(* CODESYS project xlh_gantry_00_01.project
   Description: Receives some incoming messages and echoes them with CAN-ID +1
   Company: 3S - Smart Software Solutions GmbH
   Version: 1.0.0.0
   Title: CAN Bus API Example
   Author: 3S - Smart Software Solutions GmbH

Project tree, tasks and I/O mapping:
  xLH_base : CODESYS Control for Raspberry Pi 64 SL, CODESYS, order no. 2302000009, version 4.18.0.0
    application app
      libraries: Standard, 3.5.18.0 (System); Util, 3.5.21.0 (System); VisuDialogs, * (System); Memory, * (3S - Smart Software Solutions GmbH); CmpBitmapPool, * (System); CAN API, 1.0.0.4 (CODESYS); MemoryUtils, * (3S - Smart Software Solutions GmbH); CAA CiA 405, 4.3.0.0 (CODESYS)
      task CAN_OPEN_TASK (cyclic, interval 1 ms, priority 0) calls nothing
      task VISU_TASK (cyclic, interval 100 ms, priority 31) calls VisuElems.Visu_Prg
      task MAIN_TASK (cyclic, interval 4 ms, priority 1) calls io, MAIN_CALLER
      task SoftMotion_PlanningTask (cyclic, interval t#2ms, priority 15) calls nothing
      program MAIN_CALLER [ST]
      function block FB_SDO_READ_4_BYTE [ST]
      trace Trace_AxY (task MAIN_TASK): y_axis.fActPosition, y_axis.fSetPosition, y_axis.fSetAcceleration, y_axis.fActAcceleration, y_axis.fSetVelocity, y_axis.fActVelocity
      visualisation Visualization
      trace Trace (task MAIN_TASK): MC.diPosition, MC.iSetSpeed, MC.iDebug2Pos, MC.iDebug1Mileage, MC.auiUltrasonic[1], MC.fbReadStatusLoopTime.udiValue, MC.iSpeed2, MC.iSpeed1, MC.iPitch
      data type MOTION_CONTROL_BYTE
      MOTION_BASE/
        function block FB_XLH_MOTION_AXIS_SIMPLE_ES [ST]: mRead
        function block FB_PLC_OPEN_AXIS [ST]: plcOpen, executeToFalse
        function block FB_XLH_MOTION_AXIS_SIMPLE [ST]
        function block FB_XLH_MOTION_AXIS_BASE [ST]: mRead, mWrite
      IO/
        function block FB_XLH_GPIO [CFC]
        program io [ST]
        function block FB_XLH_DXL_RGB [CFC]
      program MC [ST]: write, read, axSmExecuteToFalse
      axis group AxisGroup: TRAFO.Kin_Gantry3, axes x_axis, y_axis, z_axis
    CANbus : CANbus, CODESYS, version 4.3.0.0
        settings: Baudrate = 1000 kbit/s
      CANopen_Manager : CANopen_Manager, CODESYS, version 4.3.0.0
          settings: NMT Start All = TRUE; Polling of optional slaves = FALSE; ConfigVersion = 50659584
        xlh_dynamixel_rgb : xlh_stamp_dynamixel_rgb, xemax ag, order no. 0, version Revision=16#00000001, FileVersion=1.0 (disabled)
            settings: NODEIDSAVED = 2; SDO Timeout = 1000000; PDO_Autoconfig = FALSE; EXPERTSETTINGS = FALSE; PDO 16#1400.COBID = 16#00000202; Process by CANopenManager = TRUE; PDO 16#1401.COBID = 16#00000302; Process by CANopenManager = TRUE; PDO 16#1402.COBID = 16#00000402; Process by CANopenManager = TRUE; PDO 16#1800.COBID = 16#00000182; Process by CANopenManager = TRUE; Dxl 1 Control.Subindex = 16#01; Dxl 1 Position.Subindex = 16#02; Dxl 1 Velocity.Subindex = 16#03; Dxl 2 Control.Subindex = 16#04; Dxl 2 Position.Subindex = 16#05; Dxl 2 Velocity.Subindex = 16#06; RGB red.Subindex = 16#01; RGB green.Subindex = 16#02; RGB blue.Subindex = 16#03; Dxl 1  Position read.Subindex = 16#01; Dxl 1 Current read.Subindex = 16#02; Dxl 2  Position read.Subindex = 16#03; Dxl 2 Current read.Subindex = 16#04; SDO List.Set COB-ID sync.Index = 16#1005; SDO List.Set COB-ID sync.Subindex = 16#00; SDO List.Set COB-ID sync.Value = 16#00000080; SDO List.Set COB-ID sync.Size = 32; SDO List.Set COB-ID sync.AbortIfError = FALSE; SDO List.Set COB-ID sync.JumpToLine = FALSE; SDO List.Set COB-ID sync.Line = 0; SDO List.Set communication cycle period.Index = 16#1006; SDO List.Set communication cycle period.Subindex = 16#00; SDO List.Set communication cycle period.Value = 16#00000000; SDO List.Set communication cycle period.Size = 32; SDO List.Set communication cycle period.AbortIfError = FALSE; SDO List.Set communication cycle period.JumpToLine = FALSE; SDO List.Set communication cycle period.Line = 0; SDO List.Set Guardtime.Index = 16#100C;
              SDO List.Set Guardtime.Subindex = 16#00; SDO List.Set Guardtime.Value = 16#000000C8; SDO List.Set Guardtime.Size = 16; SDO List.Set Guardtime.AbortIfError = FALSE; SDO List.Set Guardtime.JumpToLine = FALSE; SDO List.Set Guardtime.Line = 0; SDO List.Set Lifetime.Index = 16#100D; SDO List.Set Lifetime.Subindex = 16#00; SDO List.Set Lifetime.Value = 16#00000003; SDO List.Set Lifetime.Size = 8; SDO List.Set Lifetime.AbortIfError = FALSE; SDO List.Set Lifetime.JumpToLine = FALSE; SDO List.Set Lifetime.Line = 0; SDO List.Set Heartbeat Consumer.Index = 16#1016; SDO List.Set Heartbeat Consumer.Subindex = 16#01; SDO List.Set Heartbeat Consumer.Value = 0; SDO List.Set Heartbeat Consumer.Size = 32; SDO List.Set Heartbeat Consumer.AbortIfError = FALSE; SDO List.Set Heartbeat Consumer.JumpToLine = FALSE; SDO List.Set Heartbeat Consumer.Line = 0; SDO List.Disable PDO.Index = 16#1400; SDO List.Disable PDO.Subindex = 16#01; SDO List.Disable PDO.Value = 16#80000202; SDO List.Disable PDO.Size = 32; SDO List.Disable PDO.AbortIfError = FALSE; SDO List.Disable PDO.JumpToLine = FALSE; SDO List.Disable PDO.Line = 0; SDO List.Set transmission type.Index = 16#1400; SDO List.Set transmission type.Subindex = 16#02; SDO List.Set transmission type.Value = 16#FF; SDO List.Set transmission type.Size = 8; SDO List.Set transmission type.AbortIfError = FALSE; SDO List.Set transmission type.JumpToLine = FALSE; SDO List.Set transmission type.Line = 0; SDO List.Set and enable COB-ID.Index = 16#1400; SDO List.Set and enable COB-ID.Subindex = 16#01; SDO List.Set and enable COB-ID.Value = 16#00000202; SDO List.Set and enable COB-ID.Size = 32; SDO List.Set and enable COB-ID.AbortIfError = FALSE; SDO List.Set and enable COB-ID.JumpToLine = FALSE;
              SDO List.Set and enable COB-ID.Line = 0; SDO List.Disable PDO.Index = 16#1401; SDO List.Disable PDO.Subindex = 16#01; SDO List.Disable PDO.Value = 16#80000302; SDO List.Disable PDO.Size = 32; SDO List.Disable PDO.AbortIfError = FALSE; SDO List.Disable PDO.JumpToLine = FALSE; SDO List.Disable PDO.Line = 0; SDO List.Set transmission type.Index = 16#1401; SDO List.Set transmission type.Subindex = 16#02; SDO List.Set transmission type.Value = 16#FF; SDO List.Set transmission type.Size = 8; SDO List.Set transmission type.AbortIfError = FALSE; SDO List.Set transmission type.JumpToLine = FALSE; SDO List.Set transmission type.Line = 0; SDO List.Set and enable COB-ID.Index = 16#1401; SDO List.Set and enable COB-ID.Subindex = 16#01; SDO List.Set and enable COB-ID.Value = 16#00000302; SDO List.Set and enable COB-ID.Size = 32; SDO List.Set and enable COB-ID.AbortIfError = FALSE; SDO List.Set and enable COB-ID.JumpToLine = FALSE; SDO List.Set and enable COB-ID.Line = 0; SDO List.Disable PDO.Index = 16#1402; SDO List.Disable PDO.Subindex = 16#01; SDO List.Disable PDO.Value = 16#80000402; SDO List.Disable PDO.Size = 32; SDO List.Disable PDO.AbortIfError = FALSE; SDO List.Disable PDO.JumpToLine = FALSE; SDO List.Disable PDO.Line = 0; SDO List.Set transmission type.Index = 16#1402; SDO List.Set transmission type.Subindex = 16#02; SDO List.Set transmission type.Value = 16#FF; SDO List.Set transmission type.Size = 8; SDO List.Set transmission type.AbortIfError = FALSE; SDO List.Set transmission type.JumpToLine = FALSE; SDO List.Set transmission type.Line = 0; SDO List.Set and enable COB-ID.Index = 16#1402; SDO List.Set and enable COB-ID.Subindex = 16#01; SDO List.Set and enable COB-ID.Value = 16#00000402; SDO List.Set and enable COB-ID.Size = 32;
              SDO List.Set and enable COB-ID.AbortIfError = FALSE; SDO List.Set and enable COB-ID.JumpToLine = FALSE; SDO List.Set and enable COB-ID.Line = 0; SDO List.Disable PDO.Index = 16#1800; SDO List.Disable PDO.Subindex = 16#01; SDO List.Disable PDO.Value = 16#80000182; SDO List.Disable PDO.Size = 32; SDO List.Disable PDO.AbortIfError = FALSE; SDO List.Disable PDO.JumpToLine = FALSE; SDO List.Disable PDO.Line = 0; SDO List.Set transmission type.Index = 16#1800; SDO List.Set transmission type.Subindex = 16#02; SDO List.Set transmission type.Value = 16#FF; SDO List.Set transmission type.Size = 8; SDO List.Set transmission type.AbortIfError = FALSE; SDO List.Set transmission type.JumpToLine = FALSE; SDO List.Set transmission type.Line = 0; SDO List.Set inhibit time.Index = 16#1800; SDO List.Set inhibit time.Subindex = 16#03; SDO List.Set inhibit time.Value = 16#0000; SDO List.Set inhibit time.Size = 16; SDO List.Set inhibit time.AbortIfError = FALSE; SDO List.Set inhibit time.JumpToLine = FALSE; SDO List.Set inhibit time.Line = 0; SDO List.Set event time.Index = 16#1800; SDO List.Set event time.Subindex = 16#05; SDO List.Set event time.Value = 16#0000; SDO List.Set event time.Size = 16; SDO List.Set event time.AbortIfError = FALSE; SDO List.Set event time.JumpToLine = FALSE; SDO List.Set event time.Line = 0; SDO List.Set and enable COB-ID.Index = 16#1800; SDO List.Set and enable COB-ID.Subindex = 16#01; SDO List.Set and enable COB-ID.Value = 16#00000182; SDO List.Set and enable COB-ID.Size = 32; SDO List.Set and enable COB-ID.AbortIfError = FALSE; SDO List.Set and enable COB-ID.JumpToLine = FALSE; SDO List.Set and enable COB-ID.Line = 0; ConfigVersion = 50659584
            output app.io.dxlRgb.bDxl1Torque : BOOL  // Dxl 1 Control.Bit0
            output app.io.dxlRgb.bDxl1Led : BOOL  // Dxl 1 Control.Bit1
            output app.io.dxlRgb.uiDxl1Position : UINT  // Dxl 1 Position
            output app.io.dxlRgb.uiDxl1Velocity : UINT  // Dxl 1 Velocity
            output app.io.dxlRgb.bDxl2Torque : BOOL  // Dxl 2 Control.Bit0
            output app.io.dxlRgb.bDxl2Led : BOOL  // Dxl 2 Control.Bit1
            output app.io.dxlRgb.uiDxl2Position : UINT  // Dxl 2 Position
            output app.io.dxlRgb.uiDxl2Velocity : UINT  // Dxl 2 Velocity
            output app.io.dxlRgb.byRgbRed : USINT  // RGB red
            output app.io.dxlRgb.byRgbGreen : USINT  // RGB green
            output app.io.dxlRgb.byRgbBlue : USINT  // RGB blue
            input  app.io.dxlRgb.uiDxl1PositionGet : UINT  // Dxl 1  Position read
            input  app.io.dxlRgb.iDxl1CurrentGet : INT  // Dxl 1 Current read
            input  app.io.dxlRgb.uiDxl2PositionGet : UINT  // Dxl 2  Position read
            input  app.io.dxlRgb.iDxl2CurrentGet : INT  // Dxl 2 Current read
            unmapped channels: Dxl 1 Control, Dxl 2 Control
        xlh_motion : xlh_motion, xemax ag, order no. 0, version Revision=16#00000001, FileVersion=1.0
            settings: NODEIDSAVED = 1; SDO Timeout = 1000000; PDO_Autoconfig = FALSE; EXPERTSETTINGS = True; PDO 16#1400.COBID = 16#00000201; Process by CANopenManager = TRUE; PDO 16#1401.COBID = 16#00000301; Process by CANopenManager = TRUE; PDO 16#1402.COBID = 16#00000401; Process by CANopenManager = TRUE; PDO 16#1403.COBID = 16#00000501; Process by CANopenManager = TRUE; PDO 16#1800.COBID = 16#00000181; Process by CANopenManager = TRUE; PDO 16#1801.COBID = 16#00000281; Process by CANopenManager = TRUE; PDO 16#1802.COBID = 16#00000381; Process by CANopenManager = TRUE; Control 1.Subindex = 16#01; Control 2.Subindex = 16#02; Control 3.Subindex = 16#03; Control 4.Subindex = 16#04; Outputs 0-7.Subindex = 16#01; Outputs 8-15.Subindex = 16#02; Magnet Duty Cycle.Subindex = 16#01; Freqeuncy 1.Subindex = 16#05; Freqeuncy 2.Subindex = 16#06; Freqeuncy 3.Subindex = 16#07; Freqeuncy 4.Subindex = 16#08; Servo 1.Subindex = 16#01; Servo 2.Subindex = 16#02; Servo 3.Subindex = 16#03; Servo 4.Subindex = 16#04; Servo 5.Subindex = 16#05; Servo 6.Subindex = 16#06; Servo 7.Subindex = 16#07; Servo 8.Subindex = 16#08; Position 1.Subindex = 16#01; Position 2.Subindex = 16#02; Position 3.Subindex = 16#03;
              Position 4.Subindex = 16#04; Inputs 0-7.Subindex = 16#01; Inputs 8-15.Subindex = 16#02; Inputs CLK.Subindex = 16#03; SDO List.Set COB-ID sync.Index = 16#1005; SDO List.Set COB-ID sync.Subindex = 16#00; SDO List.Set COB-ID sync.Value = 16#00000080; SDO List.Set COB-ID sync.Size = 32; SDO List.Set COB-ID sync.AbortIfError = FALSE; SDO List.Set COB-ID sync.JumpToLine = FALSE; SDO List.Set COB-ID sync.Line = 0; SDO List.Set communication cycle period.Index = 16#1006; SDO List.Set communication cycle period.Subindex = 16#00; SDO List.Set communication cycle period.Value = 16#00000000; SDO List.Set communication cycle period.Size = 32; SDO List.Set communication cycle period.AbortIfError = FALSE; SDO List.Set communication cycle period.JumpToLine = FALSE; SDO List.Set communication cycle period.Line = 0; SDO List.Set Guardtime.Index = 16#100C; SDO List.Set Guardtime.Subindex = 16#00; SDO List.Set Guardtime.Value = 16#000000C8; SDO List.Set Guardtime.Size = 16; SDO List.Set Guardtime.AbortIfError = FALSE; SDO List.Set Guardtime.JumpToLine = FALSE; SDO List.Set Guardtime.Line = 0; SDO List.Set Lifetime.Index = 16#100D; SDO List.Set Lifetime.Subindex = 16#00; SDO List.Set Lifetime.Value = 16#00000003; SDO List.Set Lifetime.Size = 8; SDO List.Set Lifetime.AbortIfError = FALSE; SDO List.Set Lifetime.JumpToLine = FALSE; SDO List.Set Lifetime.Line = 0; SDO List.Set Heartbeat Consumer.Index = 16#1016; SDO List.Set Heartbeat Consumer.Subindex = 16#01; SDO List.Set Heartbeat Consumer.Value = 0; SDO List.Set Heartbeat Consumer.Size = 32; SDO List.Set Heartbeat Consumer.AbortIfError = FALSE; SDO List.Set Heartbeat Consumer.JumpToLine = FALSE; SDO List.Set Heartbeat Consumer.Line = 0; SDO List.Disable PDO.Index = 16#1400;
              SDO List.Disable PDO.Subindex = 16#01; SDO List.Disable PDO.Value = 16#80000201; SDO List.Disable PDO.Size = 32; SDO List.Disable PDO.AbortIfError = FALSE; SDO List.Disable PDO.JumpToLine = FALSE; SDO List.Disable PDO.Line = 0; SDO List.Set transmission type.Index = 16#1400; SDO List.Set transmission type.Subindex = 16#02; SDO List.Set transmission type.Value = 16#FF; SDO List.Set transmission type.Size = 8; SDO List.Set transmission type.AbortIfError = FALSE; SDO List.Set transmission type.JumpToLine = FALSE; SDO List.Set transmission type.Line = 0; SDO List.Set and enable COB-ID.Index = 16#1400; SDO List.Set and enable COB-ID.Subindex = 16#01; SDO List.Set and enable COB-ID.Value = 16#00000201; SDO List.Set and enable COB-ID.Size = 32; SDO List.Set and enable COB-ID.AbortIfError = FALSE; SDO List.Set and enable COB-ID.JumpToLine = FALSE; SDO List.Set and enable COB-ID.Line = 0; SDO List.Disable PDO.Index = 16#1401; SDO List.Disable PDO.Subindex = 16#01; SDO List.Disable PDO.Value = 16#80000301; SDO List.Disable PDO.Size = 32; SDO List.Disable PDO.AbortIfError = FALSE; SDO List.Disable PDO.JumpToLine = FALSE; SDO List.Disable PDO.Line = 0; SDO List.Set transmission type.Index = 16#1401; SDO List.Set transmission type.Subindex = 16#02; SDO List.Set transmission type.Value = 16#FF; SDO List.Set transmission type.Size = 8; SDO List.Set transmission type.AbortIfError = FALSE; SDO List.Set transmission type.JumpToLine = FALSE; SDO List.Set transmission type.Line = 0; SDO List.Set and enable COB-ID.Index = 16#1401; SDO List.Set and enable COB-ID.Subindex = 16#01; SDO List.Set and enable COB-ID.Value = 16#00000301; SDO List.Set and enable COB-ID.Size = 32; SDO List.Set and enable COB-ID.AbortIfError = FALSE; SDO List.Set and enable COB-ID.JumpToLine = FALSE;
              SDO List.Set and enable COB-ID.Line = 0; SDO List.Disable PDO.Index = 16#1402; SDO List.Disable PDO.Subindex = 16#01; SDO List.Disable PDO.Value = 16#80000401; SDO List.Disable PDO.Size = 32; SDO List.Disable PDO.AbortIfError = FALSE; SDO List.Disable PDO.JumpToLine = FALSE; SDO List.Disable PDO.Line = 0; SDO List.Set transmission type.Index = 16#1402; SDO List.Set transmission type.Subindex = 16#02; SDO List.Set transmission type.Value = 16#FF; SDO List.Set transmission type.Size = 8; SDO List.Set transmission type.AbortIfError = FALSE; SDO List.Set transmission type.JumpToLine = FALSE; SDO List.Set transmission type.Line = 0; SDO List.Set and enable COB-ID.Index = 16#1402; SDO List.Set and enable COB-ID.Subindex = 16#01; SDO List.Set and enable COB-ID.Value = 16#00000401; SDO List.Set and enable COB-ID.Size = 32; SDO List.Set and enable COB-ID.AbortIfError = FALSE; SDO List.Set and enable COB-ID.JumpToLine = FALSE; SDO List.Set and enable COB-ID.Line = 0; SDO List.Disable PDO.Index = 16#1403; SDO List.Disable PDO.Subindex = 16#01; SDO List.Disable PDO.Value = 16#80000501; SDO List.Disable PDO.Size = 32; SDO List.Disable PDO.AbortIfError = FALSE; SDO List.Disable PDO.JumpToLine = FALSE; SDO List.Disable PDO.Line = 0; SDO List.Set transmission type.Index = 16#1403; SDO List.Set transmission type.Subindex = 16#02; SDO List.Set transmission type.Value = 16#FF; SDO List.Set transmission type.Size = 8; SDO List.Set transmission type.AbortIfError = FALSE; SDO List.Set transmission type.JumpToLine = FALSE; SDO List.Set transmission type.Line = 0; SDO List.Set and enable COB-ID.Index = 16#1403; SDO List.Set and enable COB-ID.Subindex = 16#01; SDO List.Set and enable COB-ID.Value = 16#00000501; SDO List.Set and enable COB-ID.Size = 32;
              SDO List.Set and enable COB-ID.AbortIfError = FALSE; SDO List.Set and enable COB-ID.JumpToLine = FALSE; SDO List.Set and enable COB-ID.Line = 0; SDO List.Disable PDO.Index = 16#1800; SDO List.Disable PDO.Subindex = 16#01; SDO List.Disable PDO.Value = 16#80000181; SDO List.Disable PDO.Size = 32; SDO List.Disable PDO.AbortIfError = FALSE; SDO List.Disable PDO.JumpToLine = FALSE; SDO List.Disable PDO.Line = 0; SDO List.Set transmission type.Index = 16#1800; SDO List.Set transmission type.Subindex = 16#02; SDO List.Set transmission type.Value = 16#FF; SDO List.Set transmission type.Size = 8; SDO List.Set transmission type.AbortIfError = FALSE; SDO List.Set transmission type.JumpToLine = FALSE; SDO List.Set transmission type.Line = 0; SDO List.Set inhibit time.Index = 16#1800; SDO List.Set inhibit time.Subindex = 16#03; SDO List.Set inhibit time.Value = 16#0000; SDO List.Set inhibit time.Size = 16; SDO List.Set inhibit time.AbortIfError = FALSE; SDO List.Set inhibit time.JumpToLine = FALSE; SDO List.Set inhibit time.Line = 0; SDO List.Set event time.Index = 16#1800; SDO List.Set event time.Subindex = 16#05; SDO List.Set event time.Value = 16#0000; SDO List.Set event time.Size = 16; SDO List.Set event time.AbortIfError = FALSE; SDO List.Set event time.JumpToLine = FALSE; SDO List.Set event time.Line = 0; SDO List.Set and enable COB-ID.Index = 16#1800; SDO List.Set and enable COB-ID.Subindex = 16#01; SDO List.Set and enable COB-ID.Value = 16#00000181; SDO List.Set and enable COB-ID.Size = 32; SDO List.Set and enable COB-ID.AbortIfError = FALSE; SDO List.Set and enable COB-ID.JumpToLine = FALSE; SDO List.Set and enable COB-ID.Line = 0; SDO List.Disable PDO.Index = 16#1801; SDO List.Disable PDO.Subindex = 16#01;
              SDO List.Disable PDO.Value = 16#80000281; SDO List.Disable PDO.Size = 32; SDO List.Disable PDO.AbortIfError = FALSE; SDO List.Disable PDO.JumpToLine = FALSE; SDO List.Disable PDO.Line = 0; SDO List.Set transmission type.Index = 16#1801; SDO List.Set transmission type.Subindex = 16#02; SDO List.Set transmission type.Value = 16#FF; SDO List.Set transmission type.Size = 8; SDO List.Set transmission type.AbortIfError = FALSE; SDO List.Set transmission type.JumpToLine = FALSE; SDO List.Set transmission type.Line = 0; SDO List.Set inhibit time.Index = 16#1801; SDO List.Set inhibit time.Subindex = 16#03; SDO List.Set inhibit time.Value = 16#0000; SDO List.Set inhibit time.Size = 16; SDO List.Set inhibit time.AbortIfError = FALSE; SDO List.Set inhibit time.JumpToLine = FALSE; SDO List.Set inhibit time.Line = 0; SDO List.Set event time.Index = 16#1801; SDO List.Set event time.Subindex = 16#05; SDO List.Set event time.Value = 16#0000; SDO List.Set event time.Size = 16; SDO List.Set event time.AbortIfError = FALSE; SDO List.Set event time.JumpToLine = FALSE; SDO List.Set event time.Line = 0; SDO List.Set and enable COB-ID.Index = 16#1801; SDO List.Set and enable COB-ID.Subindex = 16#01; SDO List.Set and enable COB-ID.Value = 16#00000281; SDO List.Set and enable COB-ID.Size = 32; SDO List.Set and enable COB-ID.AbortIfError = FALSE; SDO List.Set and enable COB-ID.JumpToLine = FALSE; SDO List.Set and enable COB-ID.Line = 0; SDO List.Disable PDO.Index = 16#1802; SDO List.Disable PDO.Subindex = 16#01; SDO List.Disable PDO.Value = 16#80000381; SDO List.Disable PDO.Size = 32; SDO List.Disable PDO.AbortIfError = FALSE; SDO List.Disable PDO.JumpToLine = FALSE; SDO List.Disable PDO.Line = 0;
              SDO List.Set transmission type.Index = 16#1802; SDO List.Set transmission type.Subindex = 16#02; SDO List.Set transmission type.Value = 16#FF; SDO List.Set transmission type.Size = 8; SDO List.Set transmission type.AbortIfError = FALSE; SDO List.Set transmission type.JumpToLine = FALSE; SDO List.Set transmission type.Line = 0; SDO List.Set inhibit time.Index = 16#1802; SDO List.Set inhibit time.Subindex = 16#03; SDO List.Set inhibit time.Value = 16#0000; SDO List.Set inhibit time.Size = 16; SDO List.Set inhibit time.AbortIfError = FALSE; SDO List.Set inhibit time.JumpToLine = FALSE; SDO List.Set inhibit time.Line = 0; SDO List.Set event time.Index = 16#1802; SDO List.Set event time.Subindex = 16#05; SDO List.Set event time.Value = 16#0000; SDO List.Set event time.Size = 16; SDO List.Set event time.AbortIfError = FALSE; SDO List.Set event time.JumpToLine = FALSE; SDO List.Set event time.Line = 0; SDO List.Set and enable COB-ID.Index = 16#1802; SDO List.Set and enable COB-ID.Subindex = 16#01; SDO List.Set and enable COB-ID.Value = 16#00000381; SDO List.Set and enable COB-ID.Size = 32; SDO List.Set and enable COB-ID.AbortIfError = FALSE; SDO List.Set and enable COB-ID.JumpToLine = FALSE; SDO List.Set and enable COB-ID.Line = 0; ConfigVersion = 50659584
            output app.MC.abyControl[1] : USINT  // Control 1
            output app.MC.abyControl[2] : USINT  // Control 2
            output app.MC.abyControl[3] : USINT  // Control 3
            output app.MC.abyControl[4] : USINT  // Control 4
            output app.MC.abyOutputs[1] : USINT  // Outputs 0-7
            output app.MC.abyOutputs[2] : USINT  // Outputs 8-15
            output app.MC.uiMagnetDutyCycle : UINT  // Magnet Duty Cycle
            output app.MC.adiFrequency[1] : DINT  // Freqeuncy 1
            output app.MC.adiFrequency[2] : DINT  // Freqeuncy 2
            output app.MC.adiFrequency[3] : DINT  // Freqeuncy 3
            output app.MC.adiFrequency[4] : DINT  // Freqeuncy 4
            output app.MC.ausServo[1] : USINT  // Servo 1
            output app.MC.ausServo[2] : USINT  // Servo 2
            output app.MC.ausServo[3] : USINT  // Servo 3
            output app.MC.ausServo[4] : USINT  // Servo 4
            output app.MC.ausServo[5] : USINT  // Servo 5
            output app.MC.ausServo[6] : USINT  // Servo 6
            output app.MC.ausServo[7] : USINT  // Servo 7
            output app.MC.ausServo[8] : USINT  // Servo 8
            input  app.MC.adiPosition[1] : DINT  // Position 1
            input  app.MC.adiPosition[2] : DINT  // Position 2
            input  app.MC.adiPosition[3] : DINT  // Position 3
            input  app.MC.adiPosition[4] : DINT  // Position 4
            input  app.MC.abyInputs[1] : USINT  // Inputs 0-7
            input  app.MC.bAxXsw : BOOL  // Inputs 0-7.Bit0
            input  app.MC.bAxYsw : BOOL  // Inputs 0-7.Bit1
            input  app.MC.bAxZsw : BOOL  // Inputs 0-7.Bit2
            input  app.MC.bSensor : BOOL  // Inputs 0-7.Bit3
            input  app.MC.abyInputs[2] : USINT  // Inputs 8-15
            input  app.MC.abyInputs[3] : USINT  // Inputs CLK
    Camera device
      <Leer>
    GPIOs_A_B : GPIOs B+/Pi2, CODESYS, version 4.18.0.0
        input  app.io.gpio.bSw1 : BOOL  // digital inputs (GPIO0..GPIO31).Bit4
        input  app.io.gpio.bSw2 : BOOL  // digital inputs (GPIO0..GPIO31).Bit5
        input  app.io.gpio.bSw3 : BOOL  // digital inputs (GPIO0..GPIO31).Bit6
        input  app.io.gpio.bSw4 : BOOL  // digital inputs (GPIO0..GPIO31).Bit12
        input  app.io.gpio.bSw5 : BOOL  // digital inputs (GPIO0..GPIO31).Bit13
        input  app.io.gpio.bSw6 : BOOL  // digital inputs (GPIO0..GPIO31).Bit16
        input  app.io.gpio.bSw7 : BOOL  // digital inputs (GPIO0..GPIO31).Bit17
        input  app.io.gpio.bSw8 : BOOL  // digital inputs (GPIO0..GPIO31).Bit19
        output app.io.gpio.bLed1 : BOOL  // digital outputs (GPIO0..GPIO31).Bit20
        output app.io.gpio.bLed2 : BOOL  // digital outputs (GPIO0..GPIO31).Bit21
        output app.io.gpio.bLed3 : BOOL  // digital outputs (GPIO0..GPIO31).Bit22
        output app.io.gpio.bLed4 : BOOL  // digital outputs (GPIO0..GPIO31).Bit23
        output app.io.gpio.bLed5 : BOOL  // digital outputs (GPIO0..GPIO31).Bit24
        output app.io.gpio.bLed6 : BOOL  // digital outputs (GPIO0..GPIO31).Bit26
        output app.io.gpio.bLed7 : BOOL  // digital outputs (GPIO0..GPIO31).Bit27
        unmapped channels: digital inputs (GPIO0..GPIO31), digital outputs (GPIO0..GPIO31)
    I²C
    SoftMotion General Axis Pool
      x_axis : SM_Drive_PosControl, CODESYS, order no. 1805, version 4.18.0.0
          settings: dwRatioTechUnitsDenom = 101846; iRatioTechUnitsNum = 125; eRampType = 0; fSWMaxVelocity = 50; fSWMaxAcceleration = 100; fSWMaxDeceleration = 100; fSWMaxJerk = 1000; fSWLimitNegative = -1000; ScalingIncs = 814768; ScalingUnits = 1000; IsLinearMotor = TRUE; MaximumOutputVelocityInt = 40738; MinimumOutputVelocityInt = -40738; Kp = 0.005; MaxFollowingError = 1; PartVelocityPilotControl = 1; DeadTime = 1
      z_axis : SM_Drive_PosControl, CODESYS, order no. 1805, version 4.18.0.0
          settings: wDriveID = 3; dwRatioTechUnitsDenom = 101846; iRatioTechUnitsNum = -125; eRampType = 0; fSWMaxVelocity = 50; fSWMaxAcceleration = 100; fSWMaxDeceleration = 100; fSWMaxJerk = 1000; fSWLimitNegative = -1000; ScalingIncs = 814768; ScalingUnits = 1000; InvertDirection = TRUE; IsLinearMotor = TRUE; MaximumOutputVelocityInt = 40738; MinimumOutputVelocityInt = -40738; Kp = 0.005; MaxFollowingError = 1; DeadTime = 1
      y_axis : SM_Drive_PosControl, CODESYS, order no. 1805, version 4.18.0.0
          settings: wDriveID = 2; dwRatioTechUnitsDenom = 101846; iRatioTechUnitsNum = -125; eRampType = 0; fSWMaxVelocity = 50; fSWMaxAcceleration = 100; fSWMaxDeceleration = 100; fSWMaxJerk = 1000; fSWLimitNegative = -1000; ScalingIncs = 814768; ScalingUnits = 1000; InvertDirection = TRUE; IsLinearMotor = TRUE; MaximumOutputVelocityInt = 40738; MinimumOutputVelocityInt = -40738; Kp = 0.005; MaxFollowingError = 1; PartVelocityPilotControl = 1; DeadTime = 1
      a_axis : SM_Drive_PosControl, CODESYS, order no. 1805, version 4.18.0.0
          settings: wDriveID = 4; dwRatioTechUnitsDenom = 101846; iRatioTechUnitsNum = -125; eRampType = 0; fSWMaxVelocity = 50; fSWMaxAcceleration = 100; fSWMaxDeceleration = 100; fSWMaxJerk = 1000; fSWLimitNegative = -1000.0; ScalingIncs = 814768; ScalingUnits = 1000; InvertDirection = TRUE; IsLinearMotor = TRUE; MaximumOutputVelocityInt = 40738; MinimumOutputVelocityInt = -40738; Kp = 0.005; MaxFollowingError = 1; DeadTime = 1
    Onewire
    SPI
  libraries: VisuSymbols, 4.5.0.0 (System); DepictorBase, 1.2.0.0 (CODESYS)
  text list GlobalTextList
  5ce3da45-db07-42e7-a21c-a00fff4ed8f6|C:\Users\phe\Downloads\Musterloesung_FUP.PNG
*)

// xLH_base/app/MOTION_CONTROL_BYTE
TYPE MOTION_CONTROL_BYTE :
STRUCT
	bEnable: BOOL;
	bDir: BOOL;
	bReset: BOOL;
	bInverted: BOOL;
	bInMotion: BOOL;
	bMoveWithoutPulse: BOOL;
END_STRUCT
END_TYPE

// xLH_base/app/IO/io
PROGRAM io 
VAR_INPUT
	gpio: FB_XLH_GPIO;	
	dxlRgb: FB_XLH_DXL_RGB;
END_VAR
VAR	

END_VAR

END_PROGRAM

// xLH_base/app/IO/FB_XLH_GPIO
FUNCTION_BLOCK FB_XLH_GPIO
VAR_INPUT
	bLed1: BOOL;
	bLed2: BOOL;
	bLed3: BOOL;
	bLed4: BOOL;
	bLed5: BOOL;
	bLed6: BOOL;
	bLed7: BOOL;	
END_VAR
VAR_OUTPUT
	bSw1: BOOL;
	bSw2: BOOL;
	bSw3: BOOL;
	bSw4: BOOL;
	bSw5: BOOL;
	bSw6: BOOL;
	bSw7: BOOL;
	bSw8: BOOL;
END_VAR

END_FUNCTION_BLOCK

// xLH_base/app/IO/FB_XLH_DXL_RGB
FUNCTION_BLOCK FB_XLH_DXL_RGB
VAR_INPUT
	uiDxl1PositionGet: UINT;
	iDxl1CurrentGet: INT;
	uiDxl2PositionGet: UINT;
	iDxl2CurrentGet: INT;

	bDxl1Torque: BOOL;
	bDxl1Led: BOOL;
	uiDxl1Position: UINT;
	uiDxl1Velocity: UINT;
	
	bDxl2Torque: BOOL;
	bDxl2Led: BOOL;
	uiDxl2Position: UINT;
	uiDxl2Velocity: UINT;
	
	byRgbRed: BYTE;
	byRgbGreen: BYTE;
	byRgbBlue: BYTE;
END_VAR
VAR_OUTPUT

END_VAR

END_FUNCTION_BLOCK

// xLH_base/app/MAIN_CALLER
PROGRAM MAIN_CALLER
VAR
	bDevicesCoRunning: BOOL;
	fbTonDevicesCoRunning: TON := (PT:=T#250MS);
END_VAR

// Ueberwachung ob alle CAN-Open Devices im Status RUN sind
(*
fbTonDevicesCoRunning(IN:= 
	(xlh_motion.CANopenState = _3SCOS.DEVICE_STATE.OPERATIONAL) AND
	(xlh_dynamixel_rgb.CANopenState = _3SCOS.DEVICE_STATE.OPERATIONAL)	
);
*)
fbTonDevicesCoRunning(IN:= 
	(xlh_motion.CANopenState = _3SCOS.DEVICE_STATE.OPERATIONAL)
);
// falls alle Devices im Status RUN sind (inklusive Verzögerung), wird die POE MAIN aufgerufen
IF fbTonDevicesCoRunning.Q THEN
	MC();
END_IF

END_PROGRAM

// xLH_base/app/MC
PROGRAM MC
VAR_INPUT
	adiPosition: ARRAY[1..4] OF DINT;
	{attribute 'displaymode':='bin'} 
	abyInputs: ARRAY[1..3] OF BYTE;
	bAxXsw: BOOL;
	bAxYsw: BOOL;
	bAxZsw: BOOL;
	bSensor: BOOL;
	

END_VAR
VAR_OUTPUT
	{attribute 'displaymode':='bin'} 
	abyControl: ARRAY[1..4] OF BYTE;
	afFrequency: ARRAY[1..4] OF LREAL;
	adiFrequency: ARRAY[1..4] OF DINT;
	uiMagnetDutyCycle: UINT;
	abyOutputs: ARRAY[1..2] OF BYTE;
	ausServo: ARRAY[1..8] OF USINT;
	

END_VAR
VAR
	iState: DINT;	
	
	axX: FB_PLC_OPEN_AXIS := (fVel:=fVEL, fAcc:=fACC_DEC, fDec:=fACC_DEC, fJerk:=fJRK);
	axY: FB_PLC_OPEN_AXIS := (fVel:=fVEL, fAcc:=fACC_DEC, fDec:=fACC_DEC, fJerk:=fJRK);
	axZ: FB_PLC_OPEN_AXIS := (fVel:=fVEL, fAcc:=fACC_DEC, fDec:=fACC_DEC, fJerk:=fJRK);
	axA: FB_PLC_OPEN_AXIS := (fVel:=fVEL, fAcc:=fACC_DEC, fDec:=fACC_DEC, fJerk:=fJRK);

	fbXlhMotionAxisX: FB_XLH_MOTION_AXIS_SIMPLE_ES;
	fbXlhMotionAxisY: FB_XLH_MOTION_AXIS_SIMPLE_ES;
	fbXlhMotionAxisZ: FB_XLH_MOTION_AXIS_SIMPLE_ES;
	fbXlhMotionAxisA: FB_XLH_MOTION_AXIS_SIMPLE;	

	// ====================================================================
	
	aStrControl: ARRAY[1..4] OF MOTION_CONTROL_BYTE;
	byDummy: BYTE;
	usDummy: USINT;
	iDummy: INT;
	uiDummy: UINT;
	diDummy: DINT;
	udiDummy: UDINT;

	fbBlink: BLINK := (TIMEHIGH:=T#100MS, TIMELOW:=T#100MS, ENABLE:=TRUE);
	fbReadStatusRefreshTime: FB_SDO_READ_4_BYTE;
	fbReadStatusLoopTime: FB_SDO_READ_4_BYTE;
	bStartup: BOOL := TRUE;
	bDummy: BOOL;
	fDistanceTest: LREAL;
	bDummyX: BOOL;
	bDummyY: BOOL;
	bDummyZ: BOOL;
	fDummy: LREAL;
END_VAR
VAR CONSTANT
	fVEL : LREAL := 30.0;
	fVEL_HOMING : LREAL := 2.0;
    fACC_DEC : LREAL := 20.0;
    fJRK : LREAL := 100.0;	
END_VAR

byDummy := abyInputs[1];
bDummy := bSensor;
uiDummy := uiMagnetDutyCycle;

fDummy := y_axis.fActPosition;
fDummy := y_axis.fSetPosition;
fDummy := y_axis.fActVelocity;
fDummy := y_axis.fSetVelocity;
fDummy := y_axis.fActAcceleration;
fDummy := y_axis.fSetAcceleration;


IF bStartup THEN
	bStartup := FALSE;
	
	axX.pAxis := ADR(x_axis);
	axY.pAxis := ADR(y_axis);
	axZ.pAxis := ADR(z_axis);
	axA.pAxis := ADR(a_axis);

	fbXlhMotionAxisX.pfbAxisPlcOpen := ADR(axX);
	fbXlhMotionAxisX.pAxis := ADR(x_axis);
	fbXlhMotionAxisX.pbEs := ADR(bAxXsw);
	
	fbXlhMotionAxisY.pfbAxisPlcOpen := ADR(axY);
	fbXlhMotionAxisY.pAxis := ADR(y_axis);
	fbXlhMotionAxisY.pbEs := ADR(bAxYsw);

	fbXlhMotionAxisZ.pfbAxisPlcOpen := ADR(axZ);
	fbXlhMotionAxisZ.pAxis := ADR(z_axis);
	fbXlhMotionAxisZ.pbEs := ADR(bAxZsw);
	
	fbXlhMotionAxisA.pfbAxisPlcOpen := ADR(axA);
	fbXlhMotionAxisA.pAxis := ADR(a_axis);
	//fbXlhMotionAxisA.pbEs := ADR(bAxAsw);
	
	io.dxlRgb.bDxl1Torque := TRUE;
	io.dxlRgb.uiDxl1Position := 1024;
	io.dxlRgb.uiDxl1Velocity := 50;
	
	io.dxlRgb.bDxl2Torque := TRUE;
	io.dxlRgb.uiDxl2Position := 1024;
	io.dxlRgb.uiDxl2Velocity := 50;
	
	io.dxlRgb.byRgbRed := 0;
	io.dxlRgb.byRgbGreen := 0;
	io.dxlRgb.byRgbBlue := 0;
	
	ausServo[1] := 128;
END_IF

MC.read();

axX();
axY();
axZ();
axA();
fbXlhMotionAxisX();
fbXlhMotionAxisY();
fbXlhMotionAxisZ();
fbXlhMotionAxisA();



CASE iState OF
	// ============================================================================================
	// STARTUP UND INITIALISIERUNG
	// ============================================================================================
	
	0:		// Startup
		bDummyX := TRUE;
		bDummyY := TRUE;
		bDummyZ := TRUE;
		iState := 50;


	50:	// Power der Achsen
		axX.mcp.Enable := TRUE; axX.mcp.bRegulatorOn := TRUE; axX.mcp.bDriveStart := TRUE;
		axY.mcp.Enable := TRUE; axY.mcp.bRegulatorOn := TRUE; axY.mcp.bDriveStart := TRUE;
		axZ.mcp.Enable := TRUE; axZ.mcp.bRegulatorOn := TRUE; axZ.mcp.bDriveStart := TRUE;
		axA.mcp.Enable := TRUE; axA.mcp.bRegulatorOn := TRUE; axA.mcp.bDriveStart := TRUE;
		
		// https://content.helpme-codesys.com/en/libs/SM3_Basic/Current/SM3_Basic/DataTypes/DriveInterface/SMC_AXIS_STATE.html
		IF (axX.mcp.Status AND x_axis.nAxisState = SMC_AXIS_STATE.standstill) AND
		   (axY.mcp.Status AND y_axis.nAxisState = SMC_AXIS_STATE.standstill) AND
		   (axZ.mcp.Status AND z_axis.nAxisState = SMC_AXIS_STATE.standstill) AND
		   (axA.mcp.Status AND a_axis.nAxisState = SMC_AXIS_STATE.standstill) THEN
			MC.axSmExecuteToFalse();
			iState := iState + 10;
		END_IF
		
	60: 
 		iState := 100;

	100:	// Homing
		fbXlhMotionAxisX.bHoming := TRUE;
		fbXlhMotionAxisX.fVelHoming := fVEL_HOMING;
		fbXlhMotionAxisX.fVelHomingFast := 3.0 * fVEL_HOMING;
		fbXlhMotionAxisX.eMcHomingDirection := MC_DIRECTION.positive;
		fbXlhMotionAxisX.fOffset := -100.0;
		
		fbXlhMotionAxisY.bHoming := TRUE;
		fbXlhMotionAxisY.fVelHoming := fVEL_HOMING;
		fbXlhMotionAxisY.fVelHomingFast := 3.0 * fVEL_HOMING;
		fbXlhMotionAxisY.eMcHomingDirection := MC_DIRECTION.positive;
		fbXlhMotionAxisY.fOffset := -100.0;
		
		fbXlhMotionAxisZ.bHoming := TRUE;
		fbXlhMotionAxisZ.fVelHoming := fVEL_HOMING;
		fbXlhMotionAxisZ.fVelHomingFast := 3.0 * fVEL_HOMING;
		fbXlhMotionAxisZ.eMcHomingDirection := MC_DIRECTION.positive;
		fbXlhMotionAxisZ.fOffset := -30.0;
		
		fbXlhMotionAxisA.bHoming := TRUE;
		fbXlhMotionAxisA.fVelHoming := fVEL_HOMING;
		//fbXlhMotionAxisA.rVelHomingFast := 3.0 * VEL_HOMING;
		fbXlhMotionAxisA.eMcHomingDirection := MC_DIRECTION.positive;
		//fbXlhMotionAxisA.rOffset := 0.0;
		
		IF fbXlhMotionAxisX.bHomingDone AND
           fbXlhMotionAxisY.bHomingDone AND
           fbXlhMotionAxisZ.bHomingDone AND
           fbXlhMotionAxisA.bHomingDone THEN
			MC.axSmExecuteToFalse();
			fbXlhMotionAxisX.bHoming := FALSE;
			fbXlhMotionAxisY.bHoming := FALSE;
			fbXlhMotionAxisZ.bHoming := FALSE;
			fbXlhMotionAxisA.bHoming := FALSE;
			iState := iState + 10;
		END_IF	

	110: 
 		iState := 1000;

	// ============================================================================================
	// Kommandos
	// ============================================================================================
	
	1000: 	// Resetierung der Kommandos
		axX.fVel := fVEL;
		axX.fAcc := fACC_DEC;
		axX.fJerk := fJRK;
		
		axY.fVel := fVEL;
		axY.fAcc := fACC_DEC;
		axY.fJerk := fJRK;
		
		axZ.fVel := fVEL;
		axZ.fAcc := fACC_DEC;
		axZ.fJerk := fJRK;
		
		MC.axSmExecuteToFalse();
		iState := iState + 10;
		
	1010:	// warte auf Aktion		
		//IF io.gpio.bSw5 THEN iState := 2000; END_IF
		//IF io.gpio.bSw6 THEN iState := 2010; END_IF
		IF io.gpio.bSw5 THEN iState := 2020; END_IF
		IF io.gpio.bSw6 THEN iState := 2030; END_IF
		//IF io.gpio.bSw5 THEN iState := 2040; END_IF
		//IF io.gpio.bSw6 THEN iState := 2050; END_IF
		//IF io.gpio.bSw5 THEN iState := 2060; END_IF
		//IF io.gpio.bSw6 THEN iState := 2070; END_IF
		iState := 2100;
	
	2000:
		axX.mcmr.Execute := TRUE;
		axX.mcmr.Distance := 10.0;
		IF axX.mcmr.Done THEN
			iState := 1000;
		END_IF
		
	2010:
		axX.mcmr.Execute := TRUE;
		axX.mcmr.Distance := -10.0;
		IF axX.mcmr.Done THEN
			iState := 1000;
		END_IF
		
	2020:
		axY.mcmr.Execute := TRUE;
		axY.mcmr.Distance := 10.0;
		IF axY.mcmr.Done THEN
			iState := 1000;
		END_IF
		
	2030:
		axY.mcmr.Execute := TRUE;
		axY.mcmr.Distance := -10.0;
		IF axY.mcmr.Done THEN
			iState := 1000;
		END_IF
		
	2040:
		axZ.mcmr.Execute := TRUE;
		axZ.mcmr.Distance := 10.0;
		IF axZ.mcmr.Done THEN
			iState := 1000;
		END_IF
		
	2050:
		axZ.mcmr.Execute := TRUE;
		axZ.mcmr.Distance := -10.0;
		IF axZ.mcmr.Done THEN
			iState := 1000;
		END_IF
		
	2060:
		axA.mcmr.Execute := TRUE;
		axA.mcmr.Distance := 10.0;
		IF axA.mcmr.Done THEN
			iState := 1000;
		END_IF
		
	2070:
		axA.mcmr.Execute := TRUE;
		axA.mcmr.Distance := -10.0;
		IF axA.mcmr.Done THEN
			iState := 1000;
		END_IF
	
	2100:	
		fDistanceTest := 25.0;
		axX.mcma.Execute := bDummyX;
		axX.mcma.Position := fDistanceTest;
		axY.mcma.Execute := bDummyY;
		axY.mcma.Position := fDistanceTest;
		axZ.mcma.Execute := bDummyZ;
		axZ.mcma.Position := fDistanceTest;
		IF (axX.mcma.Done OR NOT bDummyX) AND (axY.mcma.Done OR NOT bDummyY) AND (axZ.mcma.Done OR NOT bDummyZ) THEN
			MC.axSmExecuteToFalse();
			iState := iState + 10;
		END_IF
		
	2110:
		iState := iState + 10;
		
	2120:
		axX.mcma.Execute := bDummyX;
		axX.mcma.Position := (-1.0)*fDistanceTest;
		axY.mcma.Execute := bDummyY;
		axY.mcma.Position := (-1.0)*fDistanceTest;
		axZ.mcma.Execute := bDummyZ;
		axZ.mcma.Position := (-1.0)*fDistanceTest;
		IF (axX.mcma.Done OR NOT bDummyX) AND (axY.mcma.Done OR NOT bDummyY) AND (axZ.mcma.Done OR NOT bDummyZ) THEN
			MC.axSmExecuteToFalse();
			iState := iState + 10;
		END_IF
		
	2130:
		iState := 2100;
		
		
		
		
		
		
		
		

END_CASE

MC.write();

usDummy := ausServo[1];
ausServo[2] := ausServo[1];
ausServo[3] := ausServo[1];
ausServo[4] := ausServo[1];
ausServo[5] := ausServo[1];
ausServo[6] := ausServo[1];
ausServo[7] := ausServo[1];
ausServo[8] := ausServo[1];

// Dynamixel + RGB
bDummy := io.dxlRgb.bDxl1Torque;
bDummy := io.dxlRgb.bDxl1Led;
uiDummy := io.dxlRgb.uiDxl1Position;
uiDummy := io.dxlRgb.uiDxl1Velocity;
uiDummy := io.dxlRgb.uiDxl1PositionGet;
iDummy := io.dxlRgb.iDxl1CurrentGet;

bDummy := io.dxlRgb.bDxl2Torque;
bDummy := io.dxlRgb.bDxl2Led;
uiDummy := io.dxlRgb.uiDxl2Position;
uiDummy := io.dxlRgb.uiDxl2Velocity;
uiDummy := io.dxlRgb.uiDxl2PositionGet;
iDummy := io.dxlRgb.iDxl2CurrentGet;

byDummy := io.dxlRgb.byRgbRed;
byDummy := io.dxlRgb.byRgbGreen;
byDummy := io.dxlRgb.byRgbBlue;



(*
IF bStartup THEN
	bStartup := FALSE;
	
	aStrControl[1].bEnable := TRUE;
	aStrControl[1].bInMotion := TRUE;
	adiFrequency[1] := 30000;
	
	ausServo[1] := 100;
	
END_IF

aStrControl[2].bEnable := aStrControl[1].bEnable;
aStrControl[3].bEnable := aStrControl[1].bEnable;
aStrControl[4].bEnable := aStrControl[1].bEnable;

aStrControl[2].bInMotion := aStrControl[1].bInMotion;
aStrControl[3].bInMotion := aStrControl[1].bInMotion;
aStrControl[4].bInMotion := aStrControl[1].bInMotion;

adiFrequency[2] := adiFrequency[1];
adiFrequency[3] := adiFrequency[1];
adiFrequency[4] := adiFrequency[1];

abyControl[1] := MEM.PackBitsToByte(
		FALSE,
		FALSE,
		aStrControl[1].bMoveWithoutPulse,
		aStrControl[1].bInMotion,
		aStrControl[1].bInverted,
		aStrControl[1].bReset,
		aStrControl[1].bDir,
		aStrControl[1].bEnable);	

abyControl[2] := MEM.PackBitsToByte(
		FALSE,
		FALSE,
		aStrControl[2].bMoveWithoutPulse,
		aStrControl[2].bInMotion,
		aStrControl[2].bInverted,
		aStrControl[2].bReset,
		aStrControl[2].bDir,
		aStrControl[2].bEnable);	
		
abyControl[3] := MEM.PackBitsToByte(
		FALSE,
		FALSE,
		aStrControl[3].bMoveWithoutPulse,
		aStrControl[3].bInMotion,
		aStrControl[3].bInverted,
		aStrControl[3].bReset,
		aStrControl[3].bDir,
		aStrControl[3].bEnable);	
		
abyControl[4] := MEM.PackBitsToByte(
		FALSE,
		FALSE,
		aStrControl[4].bMoveWithoutPulse,
		aStrControl[4].bInMotion,
		aStrControl[4].bInverted,
		aStrControl[4].bReset,
		aStrControl[4].bDir,
		aStrControl[4].bEnable);	

byDummy := abyControl[1];
byDummy := abyControl[2];
byDummy := abyControl[3];
byDummy := abyControl[4];

diDummy := adiFrequency[1];
diDummy := adiFrequency[2];
diDummy := adiFrequency[3];
diDummy := adiFrequency[4];

diDummy := adiPosition[1];
diDummy := adiPosition[2];
diDummy := adiPosition[3];
diDummy := adiPosition[4];

uiDummy := uiMagnetDutyCycle;

byDummy := abyInputs[1];
byDummy := abyInputs[2];
byDummy := abyInputs[3];

byDummy := abyOutputs[1];
byDummy := abyOutputs[2];

usDummy := ausServo[1];
ausServo[2] := ausServo[1];
ausServo[3] := ausServo[1];
ausServo[4] := ausServo[1];
ausServo[5] := ausServo[1];
ausServo[6] := ausServo[1];
ausServo[7] := ausServo[1];
ausServo[8] := ausServo[1];

// ##############################################################
// xlh_ddsm210_imu
// xlh_ddsm210_ultrasonic
fbBlink();
fbReadStatusRefreshTime(
	bEnable:=fbBlink.OUT,
	usCoDeviceId:=xlh_motion.NodeID,
	uiIndex:=16#5800, usSubindex:=1);
fbReadStatusLoopTime(
	bEnable:= NOT fbBlink.OUT,
	usCoDeviceId:=xlh_motion.NodeID,
	uiIndex:=16#5800, usSubindex:=2);
udiDummy := fbReadStatusRefreshTime.udiValue;
udiDummy := fbReadStatusLoopTime.udiValue;

// ##############################################################
*)

ACTION write:
fbXlhMotionAxisX.mWrite();
fbXlhMotionAxisY.mWrite();
fbXlhMotionAxisZ.mWrite();
fbXlhMotionAxisA.mWrite();

abyControl[1] := MEM.PackBitsToByte(
		FALSE,
		FALSE,
		fbXlhMotionAxisX.bMoveWithoutPulse,
		fbXlhMotionAxisX._bInMotion,
		fbXlhMotionAxisX.bInverted,
		fbXlhMotionAxisX.bReset,
		fbXlhMotionAxisX._bDir,
		fbXlhMotionAxisX._bEn);
afFrequency[1] := 150000000.0 / LIMIT(0.25, TO_REAL(fbXlhMotionAxisX._diFrequency), 50000.0);
adiFrequency[1] := LREAL_TO_DINT(LIMIT(2000.0, afFrequency[1], 600000000.0));

abyControl[2] := MEM.PackBitsToByte(
		FALSE,
		FALSE,
		fbXlhMotionAxisY.bMoveWithoutPulse,
		fbXlhMotionAxisY._bInMotion,
		fbXlhMotionAxisY.bInverted,
		fbXlhMotionAxisY.bReset,
		fbXlhMotionAxisY._bDir,
		fbXlhMotionAxisY._bEn);
afFrequency[2] := 150000000.0 / LIMIT(0.25, TO_REAL(fbXlhMotionAxisY._diFrequency), 50000.0);
adiFrequency[2] := LREAL_TO_DINT(LIMIT(2000.0, afFrequency[2], 600000000.0));

abyControl[3] := MEM.PackBitsToByte(
		FALSE,
		FALSE,
		fbXlhMotionAxisZ.bMoveWithoutPulse,
		fbXlhMotionAxisZ._bInMotion,
		fbXlhMotionAxisZ.bInverted,
		fbXlhMotionAxisZ.bReset,
		fbXlhMotionAxisZ._bDir,
		fbXlhMotionAxisZ._bEn);
afFrequency[3] := 150000000.0 / LIMIT(0.25, TO_REAL(fbXlhMotionAxisZ._diFrequency), 50000.0);
adiFrequency[3] := LREAL_TO_DINT(LIMIT(2000.0, afFrequency[3], 600000000.0));

abyControl[4] := MEM.PackBitsToByte(
		FALSE,
		FALSE,
		fbXlhMotionAxisA.bMoveWithoutPulse,
		fbXlhMotionAxisA._bInMotion,
		fbXlhMotionAxisA.bInverted,
		fbXlhMotionAxisA.bReset,
		fbXlhMotionAxisA._bDir,
		fbXlhMotionAxisA._bEn);
afFrequency[4] := 150000000.0 / LIMIT(0.25, TO_REAL(fbXlhMotionAxisA._diFrequency), 50000.0);
adiFrequency[4] := LREAL_TO_DINT(LIMIT(2000.0, afFrequency[4], 600000000.0));

// FixMe: frequency udint!
END_ACTION

ACTION read:
fbXlhMotionAxisX.diPosition := adiPosition[1];
fbXlhMotionAxisX.mRead();

fbXlhMotionAxisY.diPosition := adiPosition[2];
fbXlhMotionAxisY.mRead();

fbXlhMotionAxisZ.diPosition := adiPosition[3];
fbXlhMotionAxisZ.mRead();

fbXlhMotionAxisA.diPosition := adiPosition[4];
fbXlhMotionAxisA.mRead();
END_ACTION

ACTION axSmExecuteToFalse:
axX.executeToFalse();
axY.executeToFalse();
axZ.executeToFalse();
axA.executeToFalse();
END_ACTION

END_PROGRAM

// xLH_base/app/MOTION_BASE/FB_PLC_OPEN_AXIS
FUNCTION_BLOCK FB_PLC_OPEN_AXIS
VAR_INPUT	
	fVel: LREAL := 200.0;
	fAcc: LREAL := 750.0;
	fDec: LREAL := 750.0;
	fJerk: LREAL := 10000.0;
	
	mcrs: MC_ReadStatus := (Enable:=TRUE);
	mcrae: MC_ReadAxisError := (Enable:=TRUE);
	mcr: MC_Reset;
	smcrfbe: SMC_ReadFBError;
	mcp: MC_Power := (Enable:=FALSE, bRegulatorOn:=FALSE, bDriveStart:=FALSE);
	mcs: MC_Stop;
	mcma: MC_MoveAbsolute := (Velocity:=100.0, Acceleration:=1000.0, Deceleration:=1000.0, Jerk:=10000.0);
	mcmr: MC_MoveRelative := (Velocity:=100.0, Acceleration:=1000.0, Deceleration:=1000.0, Jerk:=10000.0);
	mcmv: MC_MoveVelocity := (Velocity:=100.0, Acceleration:=1000.0, Deceleration:=1000.0, Jerk:=10000.0, Direction:=-1);// 1 Positiv, -1 Negativ	
	
	pAxis: POINTER TO AXIS_REF_SM3; 
	// https://content.helpme-codesys.com/en/libs/SM3_Drive_PosControl/Current/AXIS_REF_POSCONTROL.html
	//axisPosControl: REFERENCE TO AXIS_REF_POSCONTROL;
END_VAR
VAR_OUTPUT	
	bError: BOOL;
	fActPos: LREAL;
	fActVel: LREAL;
	fActAcc: LREAL;
END_VAR
VAR
	bDummy: BOOL;
END_VAR

// Aufruf der PLC OPEN Motionbausteine
plcOpen();

// Fehlerauswertung
bError := mcs.Error OR mcmr.Error OR mcma.Error OR mcmv.Error;

// Zuweisung der Motion Control Istwerte
IF pAxis > 16#0 THEN
	fActPos := pAxis^.fActPosition;
	fActVel := pAxis^.fActVelocity;
	fActAcc := pAxis^.fActAcceleration;
END_IF

// axis.nAxisState = SMC_AXIS_STATE.standstill
// axis.nAxisState = SMC_AXIS_STATE.standstill

ACTION plcOpen:
IF pAxis > 16#0 THEN
	// Aufruf der PLC Open Motion Control Baustein
	mcrs(Axis:=pAxis^);// MC_ReadStatus https://help.codesys.com/search;version=3.5.17.0;term=MC_ReadStatus
	mcrae(Axis:=pAxis^);// MC_ReadAxisError https://help.codesys.com/webapp/ML6Svtks37sht2hVC_6YLIhf2ZY%2FMC_ReadAxisError;product=SM3_Basic;version=4.9.0.0
	mcr(Axis:=pAxis^);// MC_Reset https://help.codesys.com/webapp/xiNnxNPAb5nA4ocm6PFB_cHgUb4%2FMC_Reset;product=SM3_Basic;version=4.9.0.0
	smcrfbe(Axis:=pAxis^);// SMC_ReadFBError https://help.codesys.com/webapp/xUeuGLdUseEDKMLaPLQmdZO45P8%2FSMC_ReadFBError;product=SM3_Basic;version=4.9.0.0
	mcp(Axis:=pAxis^);// MC_Power https://help.codesys.com/webapp/xiNnxNPAb5nA4ocm6PFB_cHgUb4%2FMC_Power;product=SM3_Basic;version=4.9.0.0
	//mch(Axis:=pAxis^);// MC_Home https://content.helpme-codesys.com/en/libs/SM3_Basic/Current/SM3_Basic/POUs/Movement/MC_Home.html
	
	mcs.Deceleration := fDec;
	mcs.Jerk := fJerk;
	mcs(Axis:=pAxis^);// MC_Stop https://help.codesys.com/webapp/xUeuGLdUseEDKMLaPLQmdZO45P8%2FSMC_ReadFBError;product=SM3_Basic;version=4.9.0.0
	
	mcma.Velocity := fVel;
	mcma.Acceleration := fVel;
	mcma.Deceleration := fDec;
	mcma.Jerk := fJerk;
	mcma(Axis:=pAxis^);// MC_MoveAbsolute https://help.codesys.com/webapp/74YgxSD47ycAkED81whSoB9i6wQ%2FMC_MoveAbsolute;product=SM3_Basic;version=4.9.0.0
	
	mcmr.Velocity := fVel;
	mcmr.Acceleration := fAcc;
	mcmr.Deceleration := fDec;
	mcmr.Jerk := fJerk;
	mcmr(Axis:=pAxis^);// MC_MoveRelative https://help.codesys.com/webapp/74YgxSD47ycAkED81whSoB9i6wQ%2FMC_MoveRelative;product=SM3_Basic;version=4.9.0.0
	
	mcmv.Velocity := fVel;
	mcmv.Acceleration := fAcc;
	mcmv.Deceleration := fDec;
	mcmv.Jerk := fJerk;
	mcmv(Axis:=pAxis^);// MC_MoveVelocity https://help.codesys.com/webapp/74YgxSD47ycAkED81whSoB9i6wQ%2FMC_MoveVelocity;product=SM3_Basic;version=4.9.0.0
	
	// SoftMotion: https://help.codesys.com/webapp/_sm_components;product=codesys_softmotion;version=4.10.0.0
	// Drive: https://help.codesys.com/webapp/_sm_inserting_connected_drive_devices;product=codesys_softmotion;version=4.10.0.0
	// SMC Error: https://help.codesys.com/webapp/4icXWiTEEU7jfvlz7ATrx-Bu-fs%2FSMC_ERROR;product=SM3_Basic;version=4.0.0.0
END_IF
END_ACTION

ACTION executeToFalse:
mcr.Execute := FALSE;
mcs.Execute := FALSE;
mcma.Execute := FALSE;
mcmr.Execute := FALSE;
mcmv.Execute := FALSE;

bDummy := mcrs.Error; 
bDummy := mcrae.Error;
bDummy := mcr.Error;
bDummy := mcp.Error;
bDummy := mcs.Error;
bDummy := mcma.Error;
bDummy := mcmr.Error;
bDummy := mcmv.Error;
END_ACTION

END_FUNCTION_BLOCK

// xLH_base/app/MOTION_BASE/FB_XLH_MOTION_AXIS_SIMPLE_ES
FUNCTION_BLOCK FB_XLH_MOTION_AXIS_SIMPLE_ES EXTENDS FB_XLH_MOTION_AXIS_BASE
VAR_INPUT
	bHoming: BOOL;
	fVelHoming: LREAL;
	fVelHomingFast: LREAL;
	eMcHomingDirection: MC_Direction;
	fOffset: LREAL;
	
	pfbAxisPlcOpen: POINTER TO FB_PLC_OPEN_AXIS;
	pbEs: POINTER TO BOOL;
END_VAR
VAR_OUTPUT
	bHomingDone: BOOL;
	bEs: BOOL;
END_VAR
VAR
	iState: INT;
	fbTonDelay1: TON;
END_VAR
VAR CONSTANT
	rOFFSET_HOMING: real := 3.0;
END_VAR

SUPER^();
bReset := FALSE; 
bMoveWithoutPulse := FALSE; 
bHomingDone := FALSE;
IF NOT bHoming THEN
	iState := 0;
END_IF

IF pfbAxisPlcOpen > 16#0 THEN
	CASE iState OF
		0: 		IF bHoming THEN
					iState := 100;	
				END_IF
				
		100:	pfbAxisPlcOpen^.fVel := fVelHomingFast;
				pfbAxisPlcOpen^.mcmv.Execute := TRUE;
				pfbAxisPlcOpen^.mcmv.Direction := eMcHomingDirection;
				IF NOT bEs THEN
					pfbAxisPlcOpen^.executeToFalse();
					iState := iState + 10;
				END_IF
				
		110:	pfbAxisPlcOpen^.mcs.Execute := TRUE;
				IF pfbAxisPlcOpen^.mcs.Done THEN
					pfbAxisPlcOpen^.executeToFalse();
					iState := iState + 10;
				END_IF
				
				
		120:	pfbAxisPlcOpen^.mcmr.Execute := TRUE;
				pfbAxisPlcOpen^.fVel := fVelHoming;
				IF eMcHomingDirection = MC_DIRECTION.negative THEN
					pfbAxisPlcOpen^.mcmr.Distance := rOFFSET_HOMING;
				ELSE
					pfbAxisPlcOpen^.mcmr.Distance := (-1.0) * rOFFSET_HOMING;
				END_IF
				IF pfbAxisPlcOpen^.mcmr.Done THEN
					pfbAxisPlcOpen^.executeToFalse();
					iState := iState + 10;
				END_IF
				
		130:	pfbAxisPlcOpen^.fVel := fVelHoming;
				pfbAxisPlcOpen^.mcmv.Execute := TRUE;
				pfbAxisPlcOpen^.mcmv.Direction := eMcHomingDirection;
				IF NOT bEs THEN
					pfbAxisPlcOpen^.executeToFalse();
					iState := iState + 10;
				END_IF
				
		140:	pfbAxisPlcOpen^.mcs.Execute := TRUE;
				IF pfbAxisPlcOpen^.mcs.Done THEN
					pfbAxisPlcOpen^.executeToFalse();
					iState := iState + 10;
				END_IF		
				
		150:	pfbAxisPlcOpen^.mcmr.Execute := TRUE;
				pfbAxisPlcOpen^.fVel := TO_REAL(pfbAxisPlcOpen^.pAxis^.fSWMaxVelocity); 
				pfbAxisPlcOpen^.mcmr.Distance := fOffset;
				IF pfbAxisPlcOpen^.mcmr.Done THEN
					pfbAxisPlcOpen^.executeToFalse();
					iState := iState + 10;
				END_IF
				
		160:	//bReset := TRUE; 
				bMoveWithoutPulse := TRUE; 
				pfbAxisPlcOpen^.mcma.Execute := TRUE;
				pfbAxisPlcOpen^.fVel := TO_REAL(pfbAxisPlcOpen^.pAxis^.fSWMaxVelocity); 
				pfbAxisPlcOpen^.mcma.Position := 0.0;
				IF pfbAxisPlcOpen^.mcma.Done THEN
					pfbAxisPlcOpen^.executeToFalse();
					iState := iState + 10;
				END_IF
				
		170:	//bReset := TRUE; 
				bMoveWithoutPulse := TRUE; 
				fbTonDelay1.IN := TRUE;
				fbTonDelay1.PT := T#250MS;
				IF fbTonDelay1.Q THEN
					iState := iState + 10;
				END_IF
		
		180: 	bHomingDone := TRUE;
		
		ELSE 	iState := 0;
	END_CASE
ELSE
	iState := 0;
END_IF

fbTonDelay1();
fbTonDelay1.IN := FALSE;

METHOD mRead : BOOL
VAR_INPUT
END_VAR
VAR

END_VAR
SUPER^.mRead();
IF pbEs > 16#0 THEN
	bEs := pbEs^;
ELSE
	bEs := FALSE;
END_IF
END_METHOD

END_FUNCTION_BLOCK

// xLH_base/app/MOTION_BASE/FB_XLH_MOTION_AXIS_BASE
FUNCTION_BLOCK FB_XLH_MOTION_AXIS_BASE
VAR_INPUT
	bInverted: BOOL;
	bReset: BOOL;
	bMoveWithoutPulse: BOOL;
	pAxis: POINTER TO AXIS_REF_POSCONTROL;
	diPosition: DINT;
END_VAR
VAR_OUTPUT
	
END_VAR
VAR
	_fbTofSm1: TOF;
	_bEn: BOOL;
	_bDir: BOOL;
	_bInMotion: BOOL;
	_diFrequency: DINT;	
END_VAR

METHOD mRead : BOOL
VAR_INPUT
END_VAR
VAR

END_VAR
IF pAxis > 16#0 THEN
	pAxis^.in.dwActPosition := TO_DWORD(diPosition);
	pAxis^.in.bDriveStartRealState := TRUE;
	pAxis^.in.bRegulatorRealState := TRUE;
END_IF
END_METHOD

METHOD mWrite : BOOL
VAR_INPUT
END_VAR
VAR

END_VAR
IF pAxis > 16#0 THEN
	_bDir := (pAxis^.out.diSetVelocity >= 0);
	_diFrequency := ABS(pAxis^.out.diSetVelocity);
	// https://content.helpme-codesys.com/en/libs/SM3_Basic/Current/SM3_Basic/DataTypes/DriveInterface/SMC_AXIS_STATE.html
	_bEn := (pAxis^.nAxisState >= 1);
	_fbTofSm1(IN:=(pAxis^.nAxisState >= 4), PT:=T#100MS, Q=>_bInMotion);
END_IF
END_METHOD

END_FUNCTION_BLOCK

// xLH_base/app/MOTION_BASE/FB_XLH_MOTION_AXIS_SIMPLE
FUNCTION_BLOCK FB_XLH_MOTION_AXIS_SIMPLE EXTENDS FB_XLH_MOTION_AXIS_BASE
VAR_INPUT
	bHoming: BOOL;
	fVelHoming: LREAL;
	eMcHomingDirection: MC_Direction;
	
	pfbAxisPlcOpen: POINTER TO FB_PLC_OPEN_AXIS;
END_VAR
VAR_OUTPUT
	bHomingDone: BOOL;
END_VAR
VAR
	iState: INT;
	fbTonDelay1: TON;
END_VAR

SUPER^();
bReset := FALSE; 
bMoveWithoutPulse := FALSE; 
bHomingDone := FALSE;
IF NOT bHoming THEN
	iState := 0;
END_IF

IF pfbAxisPlcOpen > 16#0 THEN
	CASE iState OF
		0: 		IF bHoming THEN
					iState := 100;	
				END_IF
						
		100:	bReset := TRUE; 
				bMoveWithoutPulse := TRUE; 
				pfbAxisPlcOpen^.mcma.Execute := TRUE;
				pfbAxisPlcOpen^.fVel := fVelHoming * 10.0; 
				pfbAxisPlcOpen^.mcma.Position := 0.0;
				IF pfbAxisPlcOpen^.mcma.Done THEN
					pfbAxisPlcOpen^.executeToFalse();
					iState := iState + 10;
				END_IF
				
		110:	bReset := TRUE; 
				bMoveWithoutPulse := TRUE; 
				fbTonDelay1.IN := TRUE;
				fbTonDelay1.PT := T#100MS;
				IF fbTonDelay1.Q THEN
					bReset := FALSE; 
					bMoveWithoutPulse := FALSE;
					iState := iState + 10;
				END_IF
		
		120: 	bHomingDone := TRUE;
		
		ELSE 	iState := 0;
	END_CASE
ELSE
	iState := 0;
END_IF

fbTonDelay1();
fbTonDelay1.IN := FALSE;

END_FUNCTION_BLOCK

// xLH_base/app/FB_SDO_READ_4_BYTE
FUNCTION_BLOCK FB_SDO_READ_4_BYTE
VAR_INPUT
	bEnable: BOOL;
	usCoDeviceId: USINT;
	usNetId: USINT := 0;
	uiIndex: UINT;
	usSubindex: USINT;
END_VAR
VAR_OUTPUT
	bDone: BOOL;
	bError: BOOL;
	diValue: DINT;
	udiValue: UDINT;
END_VAR
VAR
	dwAbortCode : DWORD; //contains abort code in case of error
	fbSdoRead4Byte: CIA405.SDO_READ4;	
	fbRtEnable: R_TRIG;
END_VAR

fbRtEnable(CLK:=bEnable);
IF fbRtEnable.CLK THEN
	//bEnable := FALSE;
	bDone := FALSE;
	bError := FALSE;
END_IF

IF fbSdoRead4Byte.CONFIRM THEN
	//value was read without error
	// ==> Copy data from SDO read function block
	MEMUtils.MemCpy(pbyDest := ADR(diValue), pbySrc := ADR(fbSdoRead4Byte.DATA[1]), dwSize := SIZEOF(diValue));
	MEMUtils.MemCpy(pbyDest := ADR(udiValue), pbySrc := ADR(fbSdoRead4Byte.DATA[1]), dwSize := SIZEOF(udiValue));
	//==> On big endian systems: dwValue has to be swapped to CANopen byte order (= Little Endian).
	//MEMUtils.SwapLocalToIntel(pAddress := ADR(diValue), iSize := TO_INT(SIZEOF(diValue))); //function only swaps on big endian systems
	//MEMUtils.SwapLocalToIntel(pAddress := ADR(udiValue), iSize := TO_INT(SIZEOF(udiValue))); //function only swaps on big endian systems
	bDone := TRUE;
	bError := FALSE;
ELSIF fbSdoRead4Byte.ERROR <> CiA405.CANOPEN_KERNEL_ERROR.CANOPEN_KERNEL_NO_ERROR THEN
	//Error occured
	IF fbSdoRead4Byte.ERROR = CIA405.CANOPEN_KERNEL_ERROR.CANOPEN_KERNEL_OTHER_ERROR THEN
		//output error info contains abort code in little endian format
		MEMUtils.MemCpy(pbyDest := ADR(dwAbortCode), pbySrc := ADR(fbSdoRead4Byte.ERRORINFO), dwSize := SIZEOF(dwAbortCode));
		MEMUtils.SwapLocalToIntel(pAddress := ADR(dwAbortCode), iSize := TO_INT(SIZEOF(dwAbortCode))); //function only swaps on big endian systems	
	END_IF
	bDone := FALSE;
	bError := TRUE;
END_IF

fbSdoRead4Byte(
	NETWORK:= CANbus.NetId + 1, //CODESYS NetId starts by 0 (the number entered into the CANbus configurator); CiA405 NETWORK by 1; That is the reason why we have to increment it here.
	ENABLE:= fbRtEnable.CLK,
	TIMEOUT:= 0, //Timeout for SDO read in ms. Here: 0 ==> no timeout
	DEVICE:= usCoDeviceId, // NodeID of destination device
	CHANNEL:= 0, //SDO channel which should be used. 0 means auto channeling ==> the next free channel will be used. It depends on the slave which settings are working here but 0 and channel 1 is always working. 
	INDEX:= uiIndex, //object index which should be read
	SUBINDEX:= usSubindex //object sub index which should be read
);

END_FUNCTION_BLOCK

// xLH_base/app/Visualization
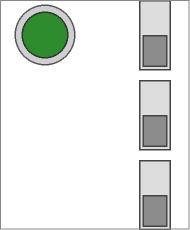
VISUALIZATION Visualization  // 190x230
    Lamp1 (10,0 70x70), variable: MC.bSensor, style: Lamp-Lamp1-Green
    DipSwitch (120,0 70x70), variable: MC.bDummyX, behaviour: TOGGLE, style: Switch-DipSwitch-Gray
    DipSwitch (120,80 70x70), variable: MC.bDummyY, behaviour: TOGGLE, style: Switch-DipSwitch-Gray
    DipSwitch (120,160 70x70), variable: MC.bDummyZ, behaviour: TOGGLE, style: Switch-DipSwitch-Gray
END_VISUALIZATION
